PROGRAM Axis_3
VAR
	bLimitPowerAxis3 AT %Q*: BOOL := TRUE;
END_VAR
VAR // added by the converter: edge detectors and wires of the graphical bodies
    _w1, _w2 : BOOL;
END_VAR

//Initial parameters of an Axis
IF _TaskInfo[fbGetCurTaskIndex.index].FirstCycle THEN
    //Initial default values:
    GVL.astAxes[3].stConfig.eHomeSeq := 1;
    GVL.astAxes[3].stConfig.fHomePosition := 0.0;
    GVL.astAxes[3].stConfig.fHomeFinishDistance := 0;
END_IF

ACT_3_Interlock();

main.stHWStatusZ.bBrakeReleased:=FALSE;  // Not used
main.stHWControlZ.bBrakeReleaseCmd:=FALSE; // Not used

// Enable Cmd from GUI
GVL.astAxes[3].stControl.bEnable:=main.stHWControlZ.bEnable;
main.stHWStatusZ.bEnabled:=GVL.astAxes[3].stStatus.bEnabled;

// Trigger Abs movement from GUI
IF main.stHWControlZ.bExecuteAbsPos  AND NOT GVL.astAxes[3].stStatus.bBusy THEN
  GVL.astAxes[3].stControl.eCommand:=E_MotionFunctions.eMoveAbsolute;
  GVL.astAxes[3].stControl.bExecute:=TRUE;
  main.stHWControlZ.bExecuteAbsPos:=FALSE;
END_IF

// Trigger Home vs LimitFwd (should be valid for all axes) from GUI
IF main.stHWControlZ.bExecuteHome  AND NOT GVL.astAxes[3].stStatus.bBusy THEN
  GVL.astAxes[3].stConfig.fHomePosition:=GVL_Parameters.fZHomePosition;
  GVL.astAxes[3].stConfig.fHomingVelFromCam:=GVL_Parameters.fZHomeVelOffCam;
  GVL.astAxes[3].stConfig.fHomingVelToCam:=GVL_Parameters.fZHomeVelToCam;
  GVL.astAxes[3].stControl.eCommand:=E_MotionFunctions.eHome;
  GVL.astAxes[3].stConfig.eHomeSeq:=E_HomingRoutines.eHomeToLimit_Fwd;
  GVL.astAxes[3].stControl.bExecute:=TRUE;
  main.stHWControlZ.bExecuteHome:=FALSE;
END_IF

//Stop Motion from GUI
IF main.stHWControlZ.bExecuteStop THEN
  GVL.astAxes[3].stControl.bStop := NOT(GVL.astAxes[3].stControl.bStop);
  GVL.astAxes[3].stControl.bExecute:=FALSE;
  main.stHWControlZ.bExecuteStop:=FALSE;
END_IF

main.stHWStatusZ.bBusy:=GVL.astAxes[3].stStatus.bBusy;
GVL.astAxes[3].stControl.bReset:=main.stHWControlZ.bExecuteReset;
main.stHWControlZ.bExecuteReset:=FALSE;
main.stHWStatusZ.bHomed:=GVL.astAxes[3].stStatus.bHomed;
main.stHWStatusZ.bHomingCmdActive:=GVL.astAxes[3].stControl.eCommand=E_MotionFunctions.eHome AND 
                                   GVL.astAxes[3].stConfig.eHomeSeq=E_HomingRoutines.eHomeToLimit_Fwd;

// Hard code velocities and acc/dec
GVL.astAxes[3].stControl.fAcceleration:=GVL_Parameters.fZStepperTargetAcc;
GVL.astAxes[3].stControl.fDeceleration:=GVL_Parameters.fZStepperTargetAcc;
GVL.astAxes[3].stControl.fVelocity:=GVL_Parameters.fZStepperTargetVelo;

// Check position is inside limits (and homed)
IF main.stHWStatusZ.bParkingRangeEnabled THEN 
  main.stHWStatusZ.bLoLoAlm:=gvl.astAxes[3].stStatus.fActPosition < GVL_Parameters.fZRangeParkL2 OR NOT main.stHWStatusZ.bHomed;
  main.stHWStatusZ.bLoAlm:=gvl.astAxes[3].stStatus.fActPosition < GVL_Parameters.fZRangeParkL1 OR NOT main.stHWStatusZ.bHomed;;
ELSE
  main.stHWStatusZ.bLoLoAlm:=gvl.astAxes[3].stStatus.fActPosition < GVL_Parameters.fZRangeL2 OR NOT main.stHWStatusZ.bHomed;;
  main.stHWStatusZ.bLoAlm:=gvl.astAxes[3].stStatus.fActPosition < GVL_Parameters.fZRangeL1 OR NOT main.stHWStatusZ.bHomed;;		
END_IF

main.stHWStatusZ.bHiAlm:=gvl.astAxes[3].stStatus.fActPosition > GVL_Parameters.fZRangeH1 OR NOT main.stHWStatusZ.bHomed;;
main.stHWStatusZ.bhiHiAlm:=gvl.astAxes[3].stStatus.fActPosition > GVL_Parameters.fZRangeH2 OR NOT main.stHWStatusZ.bHomed;;

ACTION ACT_3_Interlock:
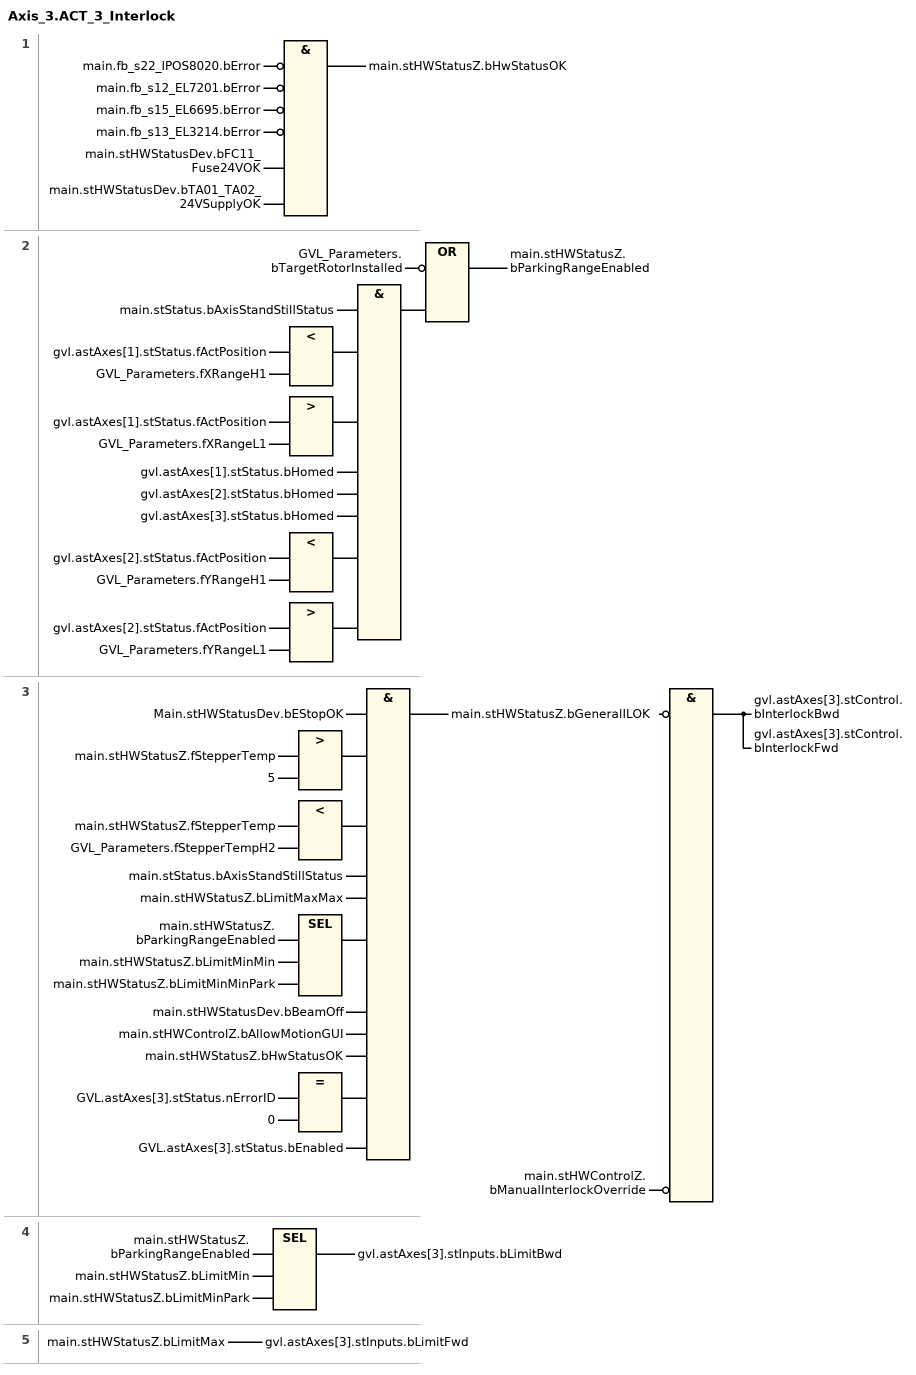
// NETWORK 1
main.stHWStatusZ.bHwStatusOK := NOT main.fb_s22_IPOS8020.bError AND NOT main.fb_s12_EL7201.bError AND NOT main.fb_s15_EL6695.bError AND NOT main.fb_s13_EL3214.bError AND main.stHWStatusDev.bFC11_Fuse24VOK AND main.stHWStatusDev.bTA01_TA02_24VSupplyOK;

// NETWORK 2
main.stHWStatusZ.bParkingRangeEnabled := NOT GVL_Parameters.bTargetRotorInstalled OR main.stStatus.bAxisStandStillStatus AND gvl.astAxes[1].stStatus.fActPosition < GVL_Parameters.fXRangeH1 AND gvl.astAxes[1].stStatus.fActPosition > GVL_Parameters.fXRangeL1 AND gvl.astAxes[1].stStatus.bHomed AND gvl.astAxes[2].stStatus.bHomed AND gvl.astAxes[3].stStatus.bHomed AND gvl.astAxes[2].stStatus.fActPosition < GVL_Parameters.fYRangeH1 AND gvl.astAxes[2].stStatus.fActPosition > GVL_Parameters.fYRangeL1;

// NETWORK 3
_w1 := Main.stHWStatusDev.bEStopOK AND main.stHWStatusZ.fStepperTemp > 5 AND main.stHWStatusZ.fStepperTemp < GVL_Parameters.fStepperTempH2 AND main.stStatus.bAxisStandStillStatus AND main.stHWStatusZ.bLimitMaxMax AND SEL(main.stHWStatusZ.bParkingRangeEnabled, main.stHWStatusZ.bLimitMinMin, main.stHWStatusZ.bLimitMinMinPark) AND main.stHWStatusDev.bBeamOff AND main.stHWControlZ.bAllowMotionGUI AND main.stHWStatusZ.bHwStatusOK AND GVL.astAxes[3].stStatus.nErrorID = 0 AND GVL.astAxes[3].stStatus.bEnabled;
main.stHWStatusZ.bGeneralILOK := _w1;
_w2 := NOT _w1 AND NOT main.stHWControlZ.bManualInterlockOverride;
gvl.astAxes[3].stControl.bInterlockBwd := _w2;
gvl.astAxes[3].stControl.bInterlockFwd := _w2;

// NETWORK 4
gvl.astAxes[3].stInputs.bLimitBwd := SEL(main.stHWStatusZ.bParkingRangeEnabled, main.stHWStatusZ.bLimitMin, main.stHWStatusZ.bLimitMinPark);

// NETWORK 5
gvl.astAxes[3].stInputs.bLimitFwd := main.stHWStatusZ.bLimitMax;

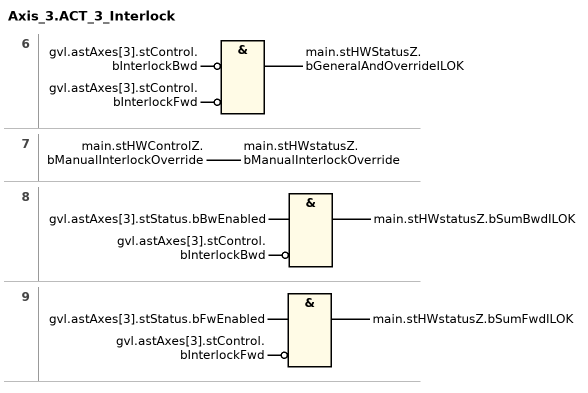
// NETWORK 6
main.stHWStatusZ.bGeneralAndOverrideILOK := NOT gvl.astAxes[3].stControl.bInterlockBwd AND NOT gvl.astAxes[3].stControl.bInterlockFwd;

// NETWORK 7
main.stHWstatusZ.bManualInterlockOverride := main.stHWControlZ.bManualInterlockOverride;

// NETWORK 8
main.stHWstatusZ.bSumBwdILOK := gvl.astAxes[3].stStatus.bBwEnabled AND NOT gvl.astAxes[3].stControl.bInterlockBwd;

// NETWORK 9
main.stHWstatusZ.bSumFwdILOK := gvl.astAxes[3].stStatus.bFwEnabled AND NOT gvl.astAxes[3].stControl.bInterlockFwd;
END_ACTION

END_PROGRAM

(* stored: Version 1.1.0.1, ProductVersion 3.1.4024.6
   POU Axis_3: Id {1bec8e22-b127-4216-8a57-916e22c1b930}, SpecialFunc None
   Action ACT_3_Interlock: Id {9a8d4546-6892-40d1-9370-4b045bf9101e} *)
